FUNCTION TryConvert_LWORD_TO_LWORD : BOOL
VAR_INPUT
	in : LWORD;
	out : REFERENCE TO LWORD;
END_VAR

out := in;
TryConvert_LWORD_TO_LWORD := TRUE;

END_FUNCTION

(* stored: Version 1.1.0.1, ProductVersion 3.1.4024.12
   POU TryConvert_LWORD_TO_LWORD: Id {bff30f7e-236c-4e4f-acea-67991c9b6666}, SpecialFunc None *)
